{attribute 'GeneratedUsingTerminal: EL4038-0000-0018'}
{attribute addProperty BoxType "EL4038-0000-0018"}
{attribute addProperty Id "EtcSlaveTerminalBaseAO_Output_Channel_1AT %Q*AO_Output_Channel_BA7EBB7C2AO_Output_Channel_2AT %Q*AO_Output_Channel_BA7EBB7C2AO_Output_Channel_3AT %Q*AO_Output_Channel_BA7EBB7C2AO_Output_Channel_4AT %Q*AO_Output_Channel_BA7EBB7C2AO_Output_Channel_5AT %Q*AO_Output_Channel_BA7EBB7C2AO_Output_Channel_6AT %Q*AO_Output_Channel_BA7EBB7C2AO_Output_Channel_7AT %Q*AO_Output_Channel_BA7EBB7C2AO_Output_Channel_8AT %Q*AO_Output_Channel_BA7EBB7C2WcStateAT %I*WcState_0B2B16F91InfoDataAT %I*InfoData_32EB74EA10"}
{attribute addProperty CRC "4163891402"}
{attribute addProperty Size "27"}
TYPE EL4038_F82FF0CA EXTENDS EtcSlaveTerminalBase :
STRUCT
	{attribute addProperty Name "AO_Output_Channel_1"}
	AO_Output_Channel_1 : AO_Output_Channel_BA7EBB7C;
	{attribute addProperty Name "AO_Output_Channel_2"}
	AO_Output_Channel_2 : AO_Output_Channel_BA7EBB7C;
	{attribute addProperty Name "AO_Output_Channel_3"}
	AO_Output_Channel_3 : AO_Output_Channel_BA7EBB7C;
	{attribute addProperty Name "AO_Output_Channel_4"}
	AO_Output_Channel_4 : AO_Output_Channel_BA7EBB7C;
	{attribute addProperty Name "AO_Output_Channel_5"}
	AO_Output_Channel_5 : AO_Output_Channel_BA7EBB7C;
	{attribute addProperty Name "AO_Output_Channel_6"}
	AO_Output_Channel_6 : AO_Output_Channel_BA7EBB7C;
	{attribute addProperty Name "AO_Output_Channel_7"}
	AO_Output_Channel_7 : AO_Output_Channel_BA7EBB7C;
	{attribute addProperty Name "AO_Output_Channel_8"}
	AO_Output_Channel_8 : AO_Output_Channel_BA7EBB7C;
	{attribute addProperty Name "WcState"}
	WcState : WcState_0B2B16F9;
	{attribute addProperty Name "InfoData"}
	InfoData : InfoData_32EB74EA;
END_STRUCT
END_TYPE

(* stored: Version 1.2.0.0, ProductVersion 3.1.4024.9
   DUT EL4038_F82FF0CA: Id {e8d0d86a-5b56-4a5f-849a-e3cc9c4acaa1} *)
